TYPE ST_Fluid :
STRUCT
END_STRUCT
END_TYPE

(* stored: Version 1.1.0.1, ProductVersion 3.1.4024.5
   DUT ST_Fluid: Id {1572871b-4263-40ef-8d4a-ead6bfbfd2d7} *)
